// TIA Portal project "LMBMD_ModbusDeviceRtu_0.0.2" (V15.1)

(* hardware
DEVICE "S7-1200 station_1"  S7-1200 Station
   slot 0: "Rack_0"  S7-1200 Rack  Rack  V1.0
   slot 1: "PLC_1"  CPU 1214C DC/DC/DC  6ES7 214-1AG40-0XB0  V4.3
   slot 3: "CB1"  CB 1241 (RS485)  6ES7 241-1CH30-1XB0  V1.0
*)

// ===== PLC "PLC_1"  CPU 1214C DC/DC/DC =====

VAR_GLOBAL   // PLC tag table "Default tag table"
   "System_Byte" AT %MB500 : Byte;
   "FirstScan" AT %M500.0 : Bool;
   "DiagStatusUpdate" AT %M500.1 : Bool;
   "AlwaysTRUE" AT %M500.2 : Bool;
   "AlwaysFALSE" AT %M500.3 : Bool;
   "System_Byte(1)" AT %MB1 : Byte;
   "System_Byte(2)" AT %MB1 : Byte;
   "Clock_Byte" AT %MB501 : Byte;
   "Clock_10Hz" AT %M501.0 : Bool;
   "Clock_5Hz" AT %M501.1 : Bool;
   "Clock_2.5Hz" AT %M501.2 : Bool;
   "Clock_2Hz" AT %M501.3 : Bool;
   "Clock_1.25Hz" AT %M501.4 : Bool;
   "Clock_1Hz" AT %M501.5 : Bool;
   "Clock_0.625Hz" AT %M501.6 : Bool;
   "Clock_0.5Hz" AT %M501.7 : Bool;
END_VAR

// folder: Example

TYPE "DeviceData"
   STRUCT
      param1 : Word;
      param2 : Word;
   END_STRUCT;
END_TYPE

// folder: LMBMD_ModbusDeviceRtu_Master

TYPE "LMBMD_ModbusDeviceRtu_RequestCfg"
// Modbus request configuration
   STRUCT
      mode : USInt := 0;   // Mode / Режим опроса
      dataAddr : UDInt := 40001;   // Starting address in the slave / Начальный адрес регистра
      len : UInt := 1;   // Data length / Длина запроса
      mapAddr : DInt := 0;   // Starting address in the read/write buffer
      enable : Bool := false;   // Заблокировать запрос / Enable request
   END_STRUCT;
END_TYPE

TYPE "LMBMD_ModbusDeviceRtu_Request"
   STRUCT
      cfg : "LMBMD_ModbusDeviceRtu_RequestCfg";
      status : "LMBMD_ModbusDeviceRtu_RequestStatus";
   END_STRUCT;
END_TYPE

TYPE "LMBMD_ModbusDeviceRtu_Data"
   STRUCT
      address : UInt;   // Modbus RTU station address
      buffer : Array[0..100] of Word;
      requests : Array[0..9] of "LMBMD_ModbusDeviceRtu_Request";
   END_STRUCT;
END_TYPE

TYPE "LMBMD_ModbusDeviceRtu_RequestStatus"
// Modbus request status
   STRUCT
      req : Bool;   // Команда на отпарвку запроса
      done : Bool;   // Опрос завершен
      busy : Bool;   // Блок в работе
      error : Bool;   // Ошибка
      status : Word;   // Статус / Error code
      errorCounter : UInt;
   END_STRUCT;
END_TYPE

TYPE "LMBMD_ModbusDeviceRtu_ComPortData"
TITLE = Настройки COM-порта
// Настройки COM-порта
   STRUCT
      port : Port := 271;   // ID порта / ID Port
      baud : UDInt := 9600;   // Скорость / Baudrate
      parity : UInt := 2;   // Паритет (0 - Нет, 1 - Нечет, 2 - Чет ) / Parity (0- None, 1 - Odd, 2 - Even)
      stopBits : UInt;   // Number of stop bits per character Valid values 1 and 2
      timeout : UInt := 500;   // Максимальное время ответа / Response timeout, ms
      status : Word;   // Статус / Response timeout
      done : Bool;   // Инициализация завершена / Execution of instruction completed without error
      error : Bool;   // Ошибка инициализации / Error
      retries : Word := 2;   // Количество повторных запросово / The number of repeated attempts by the master before the error code 0x80C8 is returned for "No response
   END_STRUCT;
END_TYPE

// folder: Example/Data

DATA_BLOCK "DataDb"   // DB1
{ S7_Optimized_Access := 'TRUE' }
VERSION : 0.1
   VAR
      device : "DeviceData";
   END_VAR
BEGIN
END_DATA_BLOCK

DATA_BLOCK "ModbusRtuMaster_DevicesDb"   // DB2
{ S7_Optimized_Access := 'TRUE' }
VERSION : 0.1
   VAR
      device1 : "LMBMD_ModbusDeviceRtu_Data";   // Device 1
      device2 : "LMBMD_ModbusDeviceRtu_Data";   // Device 2
   END_VAR
BEGIN
   device1.address := 1;
   device1.requests[0].cfg.mode := 0;
   device1.requests[0].cfg.dataAddr := 40001;
   device1.requests[0].cfg.len := 2;
   device1.requests[0].cfg.mapAddr := 0;
   device1.requests[0].cfg.enable := true;
   device1.requests[1].cfg.enable := TRUE;
   device1.requests[1].cfg.mapAddr := 1;
   device1.requests[1].cfg.len := 1;
   device2.requests[0].cfg.mapAddr := 0;
   device2.requests[0].cfg.mode := 1;
   device2.requests[0].cfg.dataAddr := 40003;
   device1.requests[1].cfg.dataAddr := 40002;
   device1.requests[1].cfg.mode := 0;
   device2.requests[0].cfg.len := 2;
   device2.address := 2;
   device2.requests[0].cfg.enable := true;
   device1.requests[9].cfg.enable := false;
   device1.requests[9].cfg.mapAddr := 0;
   device1.requests[9].cfg.len := 1;
   device1.requests[9].cfg.dataAddr := 40001;
   device1.requests[9].cfg.mode := 0;
END_DATA_BLOCK

// folder: Example/Inst

DATA_BLOCK "inst_ModbusRtu_Master"   // DB3
{ S7_Optimized_Access := 'TRUE' }
VERSION : 0.1
// stored: InstanceOfName ModbusRtu_Master
"ModbusRtu_Master"
BEGIN
END_DATA_BLOCK

// folder: LMBMD_ModbusDeviceRtu/Data

DATA_BLOCK "LMBMD_ModbusDeviceRtu_CfgDb"   // DB21
{ S7_Optimized_Access := 'TRUE' }
AUTHOR : Veshtemov
VERSION : 0.1
// Конфигурация регистров чтения по Modbus RTU
   VAR
      com : "LMBMD_ModbusDeviceRtu_ComPortData";
   END_VAR
BEGIN
   com.port := 269;
   com.baud := 9600;
   com.retries := 1;
   com.parity := 2;
   com.stopBits := 1;
END_DATA_BLOCK

DATA_BLOCK "LMBMD_ModbusDeviceRtu_DataDb"   // DB24
{ S7_Optimized_Access := 'FALSE' }
VERSION : 0.1
   VAR
      readBuffer : Array[0..255] of Byte;
      writeBuffer : Array[0..255] of Byte;
   END_VAR
BEGIN
END_DATA_BLOCK

// folder: Example

ORGANIZATION_BLOCK "Main"   // OB1, SCL, ProgramCycle
TITLE = "Main Program Sweep (Cycle)"
{ S7_Optimized_Access := 'TRUE' }
VERSION : 0.1
   VAR_INPUT
      Initial_Call : Bool;   // Initial call of this OB
      Remanence : Bool;   // =True, if remanent data are available
   END_VAR
BEGIN
   "inst_ModbusRtu_Master"(com:="LMBMD_ModbusDeviceRtu_CfgDb".com,
                           mbCommLoad:="Modbus_Comm_Load_DB",
                           mbMaster:="Modbus_Master_DB");
END_ORGANIZATION_BLOCK

// folder: Example/RS485/ModbusRtuMaster

FUNCTION_BLOCK "ModbusRtu_Master"   // FB5, SCL
{ S7_Optimized_Access := 'TRUE' }
VERSION : 0.1
// Modbus Rtu Bus
   VAR_IN_OUT
      com : "LMBMD_ModbusDeviceRtu_ComPortData";   // Serial port settings
      mbCommLoad : Modbus_Comm_Load;   // Instance of "Modbus_Comm_Load" function block
      mbMaster : Modbus_Master;   // Instance of "Modbus_Master" function block
   END_VAR
   VAR
      initTrig : R_TRIG;
      inst_LModbusDeviceRtu_Master : "LMBMD_ModbusDeviceRtu_Master";
      i : UInt;
      start : Bool;
   END_VAR
BEGIN
   // Modbus RTU Master

   REGION Serial port initialization
       IF "FirstScan" THEN
           #mbCommLoad.MODE := 4;
       END_IF;

       #mbCommLoad.RETRIES := #com.retries;

       #mbCommLoad(REQ := "FirstScan",
                   "PORT" := #com."port",
                   BAUD := #com.baud,
                   PARITY := #com.parity,
                   MB_DB := #mbMaster.MB_DB,
                   RESP_TO := #com.timeout,
                   DONE => #com.done,
                   ERROR => #com.error,
                   STATUS => #com.status);

       #initTrig(CLK := #com.done);

       IF #initTrig.Q THEN
           #i := 0;
       END_IF;
   END_REGION

   #start := NOT #inst_LModbusDeviceRtu_Master.done;

   CASE #i OF
       0:  // Device 1

           "ModbusRtu_Device1_MapData"(mdata := "ModbusRtuMaster_DevicesDb".device1,
                                       data := "DataDb".device);

           #inst_LModbusDeviceRtu_Master(start := #start,
                                         readBuffer := "LMBMD_ModbusDeviceRtu_DataDb".readBuffer,
                                         writeBuffer := "LMBMD_ModbusDeviceRtu_DataDb".writeBuffer,
                                         data := "ModbusRtuMaster_DevicesDb".device1,
                                         mbMaster := #mbMaster);

           IF #inst_LModbusDeviceRtu_Master.done THEN
               #i := #i + 1;
           END_IF;

       1:  // Device 2
           "ModbusRtu_Device2_MapData"(mdata := "ModbusRtuMaster_DevicesDb".device2,
                                       data := "DataDb".device);

           #inst_LModbusDeviceRtu_Master(start := #start,
                                         readBuffer := "LMBMD_ModbusDeviceRtu_DataDb".readBuffer,
                                         writeBuffer := "LMBMD_ModbusDeviceRtu_DataDb".writeBuffer,
                                         data := "ModbusRtuMaster_DevicesDb".device2,
                                         mbMaster := #mbMaster);

           IF #inst_LModbusDeviceRtu_Master.done THEN
               #i := #i + 1;
           END_IF;
       ELSE
           #i := 0;
   END_CASE;
END_FUNCTION_BLOCK

FUNCTION "ModbusRtu_Device2_MapData" : Void   // FC1, SCL
{ S7_Optimized_Access := 'TRUE' }
VERSION : 0.1
   VAR_IN_OUT
      mdata : "LMBMD_ModbusDeviceRtu_Data";
      data : "DeviceData";
   END_VAR
BEGIN
   // Data
   #mdata.buffer[0] := #data.param1;
   #mdata.buffer[1] := #data.param2;
END_FUNCTION

FUNCTION "ModbusRtu_Device1_MapData" : Void   // FC18, SCL
{ S7_Optimized_Access := 'TRUE' }
VERSION : 0.1
   VAR_IN_OUT
      mdata : "LMBMD_ModbusDeviceRtu_Data";
      data : "DeviceData";
   END_VAR
BEGIN
   // Data
   #data.param1 := #mdata.buffer[0];
   #data.param2 := #mdata.buffer[1];
END_FUNCTION

// folder: LMBMD_ModbusDeviceRtu/Core

FUNCTION_BLOCK "LMBMD_ModbusDeviceRtu_Master"   // FB7, SCL
{ S7_Optimized_Access := 'TRUE' }
VERSION : 0.1
   VAR_INPUT
      start : Bool;   // Пуск / Start block
   END_VAR
   VAR_OUTPUT
      busy : Bool;   // В процессе / In progress
      done : Bool;   // Окончание / Done
   END_VAR
   VAR_IN_OUT
      readBuffer : Variant;   // Буфер обмена / Pointer of read buffer (non optimized data block). For example, DB -> readBuffer: Array[0..125] of Word
      writeBuffer : Variant;   // Pointer of write buffer (non optimized data block). For example, DB -> writeBuffer: Array[0..125] of Word
      data : "LMBMD_ModbusDeviceRtu_Data";
      mbMaster : Modbus_Master;   // Instance of Modbus_Master function block
   END_VAR
   VAR
      buffer : Array[0..127] of Word;
      inst_startTrig : R_TRIG;   // Detect start
      inst_watchdogTimer : TON_TIME;   // Timer for resetting a request when unknown reason is happened
      state : USInt;   // Текущая стадия обмена / Current state
      i : Int;
      j : Int;
   END_VAR
   VAR_TEMP
      tempStart : Bool;   // Start flag
      tempRetval : Int;
      tempQntRequests : Int;   // Quantity of requests
      tempZeroIndex : DInt;
   END_VAR
   VAR CONSTANT
      STATE_STANDBY : USInt := 0;   // Ожидание / State. Standby
      STATE_SETTINGS : USInt := 1;   // Конфигурирование запроса / State. Get settings
      STATE_READ : USInt := 2;   // Запрос на чтение / State. Reading
      STATE_WRITE : USInt := 3;   // Запрос на запись / State. Writing
      STATE_HANDLE : USInt := 4;   // Обработка запроса / State. Handle results
      WATCHDOG_TIME : Time := T#10S;   // Максимальное время ожидания / Watchdog time
      ERROR_ILLEGAL_REQUEST : Word := 16#9000;   // Error. Illegal request (check request settings)
      ERROR_WATCHDOG_TIMER : Word := 16#9001;   // Error. Watchdog timer
   END_VAR
BEGIN
   #tempQntRequests := UDINT_TO_INT("LMBMD_ModbusDeviceRtu_GetArrayLength"(arr := #data.requests));
   #busy := (#state > #STATE_STANDBY); // Set busy flag

   #inst_startTrig(CLK := #start, Q => #tempStart);

   // When start go to Settings
   IF #tempStart THEN

       #done := false;
       #state := #STATE_SETTINGS;

   END_IF;

   CASE #state OF

       // Standby
       #STATE_STANDBY:

           #done := false;
           #i := 0;

       // Get request settings
       #STATE_SETTINGS:

           // With the first call we reset the counter, get the first request,
           // else we increase counter by 1 and get a next request
           IF #tempStart THEN
               #i := 0;

           ELSE
               #i := #i + 1;

               // When all requests is completed go to standby, set "done" flag 
               IF #i >= #tempQntRequests THEN
                   #done := true;
                   #state := #STATE_STANDBY;
                   RETURN;
               END_IF;
           END_IF;

           // Check request settings: we have to skip disabled or invalid requests,
           // if a request is invalid - set ERROR_ILLEGAL_REQUEST status
           FOR #j := #i TO #tempQntRequests - 1 DO

               IF NOT #data.requests[#j].cfg.enable THEN

                   #data.requests[#j].status.req := false;
                   #data.requests[#j].status.done := false;
                   #data.requests[#j].status.error := false;
                   #data.requests[#j].status.status := 0;
                   #data.requests[#j].status.errorCounter := 0;

               ELSIF NOT "LMBMD_ModbusDeviceRtu_ValidateRequest"(#data.requests[#j].cfg) THEN

                   // Set error status
                   #data.requests[#j].status.req := false;
                   #data.requests[#j].status.done := false;
                   #data.requests[#j].status.error := true;
                   #data.requests[#j].status.status := #ERROR_ILLEGAL_REQUEST;
                   #data.requests[#j].status.errorCounter := LIMIT(IN := #data.requests[#j].status.errorCounter + 1,
                                                                   MN := 0,
                                                                   MX := 65534);
               ELSE
                   #i := #j;
                   EXIT;
               END_IF;

               // When all requests is completed go to standby, set "done" flag
               IF #j = #tempQntRequests - 1 THEN
                   #done := true;
                   #state := #STATE_STANDBY;
                   RETURN;
               END_IF;

           END_FOR;

           // For writing before request we have to copy data to external write buffer
           IF #data.requests[#i].cfg.mode > 0 THEN

               // Extract data from Modbus Device to write buffer
               MOVE_BLK(IN := #data.#buffer[#data.requests[#i].cfg.mapAddr],
                        COUNT := #data.requests[#i].cfg.len,
                        OUT => #buffer[0]);

               #tempZeroIndex := 0;
               #tempRetval := Serialize(SRC_VARIABLE := #buffer,
                                        DEST_ARRAY => #writeBuffer,
                                        POS := #tempZeroIndex);

               #state := #STATE_WRITE;
           ELSE
               #state := #STATE_READ;
           END_IF;

           RETURN;

       // Read
       #STATE_READ, #STATE_WRITE:

           #data.requests[#i].status.req := true;

       // Handle results
       #STATE_HANDLE:

           #data.requests[#i].status.req := false;

           IF #data.requests[#i].status.done THEN
               #data.requests[#i].status.errorCounter := 0;

               // Copy from modbus buffer to device buffer
               IF #data.requests[#i].cfg.mode = 0 THEN

                   #tempZeroIndex := 0;
                   #tempRetval := Deserialize(SRC_ARRAY := #readBuffer,
                                              DEST_VARIABLE => #buffer,
                                              POS := #tempZeroIndex);
                   MOVE_BLK(IN := #buffer[0],
                            COUNT := #data.requests[#i].cfg.len,
                            OUT => #data.buffer[#data.requests[#i].cfg.mapAddr]);
               END_IF;

           ELSIF #data.requests[#i].status.error THEN
               #data.requests[#i].status.errorCounter := LIMIT(IN := #data.requests[#i].status.errorCounter + 1,
                                                               MN := 0,
                                                               MX := 65534);
           END_IF;

           #state := #STATE_SETTINGS;

       ELSE
           #state := #STATE_STANDBY;
   END_CASE;

   // There are different buffers for reading and writing
   IF (#state = #STATE_READ) THEN
       // Request
       #mbMaster(REQ := #data.requests[#i].status.req,
                 MB_ADDR := #data.address,
                 MODE := #data.requests[#i].cfg.mode,
                 DATA_ADDR := #data.requests[#i].cfg.dataAddr,
                 DATA_LEN := #data.requests[#i].cfg.len,
                 DONE => #data.requests[#i].status.done,
                 BUSY => #data.requests[#i].status.busy,
                 ERROR => #data.requests[#i].status.error,
                 STATUS => #data.requests[#i].status.status,
                 DATA_PTR := #readBuffer);

   ELSIF (#state = #STATE_WRITE) THEN
       // Запрос
       #mbMaster(REQ := #data.requests[#i].status.req,
                 MB_ADDR := #data.address,
                 MODE := #data.requests[#i].cfg.mode,
                 DATA_ADDR := #data.requests[#i].cfg.dataAddr,
                 DATA_LEN := #data.requests[#i].cfg.len,
                 DONE => #data.requests[#i].status.done,
                 BUSY => #data.requests[#i].status.busy,
                 ERROR => #data.requests[#i].status.error,
                 STATUS => #data.requests[#i].status.status,
                 DATA_PTR := #writeBuffer);
   END_IF;


   // Waiting response status
   IF ((#state = #STATE_READ
       OR #state = #STATE_WRITE)
       AND (#data.requests[#i].status.done
       OR #data.requests[#i].status.error))
   THEN
       #state := #STATE_HANDLE;
   END_IF;

   // Watchdog timer is needed when state stuck in Read or Write state for unknown reason,
   // in that case we set request as invalid 
   #inst_watchdogTimer(IN := (#state = #STATE_READ
                  OR #state = #STATE_WRITE),
                  PT := #WATCHDOG_TIME);

   IF #inst_watchdogTimer.Q THEN

       #data.requests[#i].status.done := false;
       #data.requests[#i].status.error := true;
       #data.requests[#i].status.status := #ERROR_WATCHDOG_TIMER;
       #data.requests[#i].status.errorCounter := LIMIT(IN := #data.requests[#i].status.errorCounter + 1,
                                                       MN := 0,
                                                       MX := 65534);

       #state := #STATE_HANDLE;

   END_IF;
END_FUNCTION_BLOCK

FUNCTION "LMBMD_ModbusDeviceRtu_ValidateRequest" : Bool   // FC2, SCL
{ S7_Optimized_Access := 'TRUE' }
VERSION : 0.1
   VAR_IN_OUT
      data : "LMBMD_ModbusDeviceRtu_RequestCfg";
   END_VAR
BEGIN
   #LMBMD_ModbusDeviceRtu_ValidateRequest :=
   #data.len > 0
   AND (#data.mode >= 0 AND #data.mode <= 2);
END_FUNCTION

FUNCTION "LMBMD_ModbusDeviceRtu_GetArrayLength" : UDInt   // FC9, SCL
{ S7_Optimized_Access := 'TRUE' }
VERSION : 0.1
   VAR_INPUT
      arr : Variant;
   END_VAR
BEGIN
   IF IS_ARRAY(#arr) THEN
       #LMBMD_ModbusDeviceRtu_GetArrayLength := CountOfElements(IN := #arr);
   ELSE
       #LMBMD_ModbusDeviceRtu_GetArrayLength := 0;
   END_IF;
END_FUNCTION

// ===== library: MasterCopy "LMB_ModbusDeviceRtu_Buffer" =====

// folder: LMB_ModbusDeviceRtu_Master

TYPE "LMB_ModbusDeviceRtu_Buffer"
// Raw data of Modbus device
   STRUCT
      readBuffer : Array[0..100] of Word;   // Read buffer
      writeBuffer : Array[0..100] of Word;   // Write buffer
   END_STRUCT;
END_TYPE

// ===== library: MasterCopy "LMB_ModbusDeviceRtu_ComPortData" =====

// folder: LMB_ModbusDeviceRtu_Master

TYPE "LMB_ModbusDeviceRtu_ComPortData"
TITLE = Настройки COM-порта
// Настройки COM-порта
   STRUCT
      port : Port := 271;   // ID порта / ID Port
      baud : UDInt := 9600;   // Скорость / Baudrate
      parity : UInt := 2;   // Паритет (0 - Нет, 1 - Нечет, 2 - Чет ) / Parity (0- None, 1 - Odd, 2 - Even)
      stopBits : UInt;   // Number of stop bits per character Valid values 1 and 2
      timeout : UInt := 500;   // Максимальное время ответа / Response timeout, ms
      status : Word;   // Статус / Response timeout
      done : Bool;   // Инициализация завершена / Execution of instruction completed without error
      error : Bool;   // Ошибка инициализации / Error
      retries : Word := 2;   // Количество повторных запросово / The number of repeated attempts by the master before the error code 0x80C8 is returned for "No response
   END_STRUCT;
END_TYPE

// ===== library: MasterCopy "LMB_ModbusDeviceRtu_Data" =====

// folder: LMB_ModbusDeviceRtu_Master

TYPE "LMB_ModbusDeviceRtu_Data"
   STRUCT
      addresss : UInt;   // Modbus RTU station address
      buffer : "LMB_ModbusDeviceRtu_Buffer";
      requests : Array[0..9] of "LMB_ModbusDeviceRtu_Request";
   END_STRUCT;
END_TYPE

// ===== library: MasterCopy "LMB_ModbusDeviceRtu_Request" =====

// folder: LMB_ModbusDeviceRtu_Master

TYPE "LMB_ModbusDeviceRtu_Request"
   STRUCT
      cfg : "LMB_ModbusDeviceRtu_RequestCfg";
      status : "LMB_ModbusDeviceRtu_RequestStatus";
   END_STRUCT;
END_TYPE

// ===== library: MasterCopy "LMB_ModbusDeviceRtu_RequestCfg" =====

// folder: LMB_ModbusDeviceRtu_Master

TYPE "LMB_ModbusDeviceRtu_RequestCfg"
// Modbus request configuration
   STRUCT
      mode : USInt := 0;   // Mode / Режим опроса
      dataAddr : UDInt := 40001;   // Starting address in the slave / Начальный адрес регистра
      len : UInt := 1;   // Data length / Длина запроса
      mapAddr : DInt := 0;   // Starting address in the read/write buffer
      enable : Bool := false;   // Заблокировать запрос / Enable request
   END_STRUCT;
END_TYPE

// ===== library: MasterCopy "LMB_ModbusDeviceRtu_RequestStatus" =====

// folder: LMB_ModbusDeviceRtu_Master

TYPE "LMB_ModbusDeviceRtu_RequestStatus"
// Modbus request status
   STRUCT
      req : Bool;   // Команда на отпарвку запроса
      done : Bool;   // Опрос завершен
      busy : Bool;   // Блок в работе
      error : Bool;   // Ошибка
      status : Word;   // Статус / Error code
      errorCounter : UInt;
   END_STRUCT;
END_TYPE

// ===== library: MasterCopy "LMB_ModbusDeviceRtu_GetArrayLength" =====

// folder: LMB_ModbusDeviceRtu_Master/Core

FUNCTION "LMB_ModbusDeviceRtu_GetArrayLength" : UDInt   // FC9, SCL
{ S7_Optimized_Access := 'TRUE' }
VERSION : 0.1
   VAR_INPUT
      arr : Variant;
   END_VAR
BEGIN
   IF IS_ARRAY(#arr) THEN
       #LMB_ModbusDeviceRtu_GetArrayLength := CountOfElements(IN := #arr);
   ELSE
       #LMB_ModbusDeviceRtu_GetArrayLength := 0;
   END_IF;
END_FUNCTION

// ===== library: MasterCopy "LMB_ModbusDeviceRtu_ValidateRequest" =====

// folder: LMB_ModbusDeviceRtu_Master/Core

FUNCTION "LMB_ModbusDeviceRtu_ValidateRequest" : Bool   // FC2, SCL
{ S7_Optimized_Access := 'TRUE' }
VERSION : 0.1
   VAR_IN_OUT
      data : "LMB_ModbusDeviceRtu_RequestCfg";
   END_VAR
BEGIN
   #LMB_ModbusDeviceRtu_ValidateRequest :=
   #data.len > 0
   AND (#data.mode >= 0 AND #data.mode <= 2);
END_FUNCTION

// ===== library: MasterCopy "LMB_ModbusDeviceRtu_Master" =====

// folder: LMB_ModbusDeviceRtu_Master/Core

FUNCTION_BLOCK "LMB_ModbusDeviceRtu_Master"   // FB7, SCL
{ S7_Optimized_Access := 'TRUE' }
VERSION : 0.1
   VAR_INPUT
      start : Bool;   // Пуск / Start block
   END_VAR
   VAR_OUTPUT
      busy : Bool;   // В процессе / In progress
      done : Bool;   // Окончание / Done
   END_VAR
   VAR_IN_OUT
      readBuffer : Variant;   // Буфер обмена / Pointer of read buffer (non optimized data block). For example, DB -> readBuffer: Array[0..125] of Word
      writeBuffer : Variant;   // Pointer of write buffer (non optimized data block). For example, DB -> writeBuffer: Array[0..125] of Word
      data : "LMB_ModbusDeviceRtu_Data";
      mbMaster : Modbus_Master;   // Instance of Modbus_Master function block
   END_VAR
   VAR
      inst_startTrig : R_TRIG;   // Detect start
      inst_watchdogTimer : TON_TIME;   // Timer for resetting a request when unknown reason is happened
      state : USInt;   // Текущая стадия обмена / Current state
      i : Int;
      j : Int;
   END_VAR
   VAR_TEMP
      tempStart : Bool;   // Start flag
      tempRetval : Int;
      tempQntRequests : Int;   // Quantity of requests
   END_VAR
   VAR CONSTANT
      STATE_STANDBY : USInt := 0;   // Ожидание / State. Standby
      STATE_SETTINGS : USInt := 1;   // Конфигурирование запроса / State. Get settings
      STATE_READ : USInt := 2;   // Запрос на чтение / State. Reading
      STATE_WRITE : USInt := 3;   // Запрос на запись / State. Writing
      STATE_HANDLE : USInt := 4;   // Обработка запроса / State. Handle results
      WATCHDOG_TIME : Time := T#10S;   // Максимальное время ожидания / Watchdog time
      ERROR_ILLEGAL_REQUEST : Word := 16#8500;   // Error. Illegal request (check request settings)
      ERROR_WATCHDOG_TIMER : Word := 16#8501;   // Error. Watchdog timer
   END_VAR
BEGIN
   #tempQntRequests := UDINT_TO_INT("LMB_ModbusDeviceRtu_GetArrayLength"(arr := #data.requests));
   #busy := (#state > #STATE_STANDBY); // Set busy flag

   #inst_startTrig(CLK := #start, Q => #tempStart);

   // When start go to Settings
   IF #tempStart THEN

       #done := false;
       #state := #STATE_SETTINGS;

   END_IF;

   CASE #state OF

       // Standby
       #STATE_STANDBY:

           #done := false;
           #i := 0;

       // Get request settings
       #STATE_SETTINGS:

           // With the first call we reset the counter, get the first request,
           // else we increase counter by 1 and get a next request
           IF #tempStart THEN
               #i := 0;

           ELSE
               #i := #i + 1;

               // When all requests is completed go to standby, set "done" flag 
               IF #i >= #tempQntRequests THEN
                   #done := true;
                   #state := #STATE_STANDBY;
                   RETURN;
               END_IF;
           END_IF;

           // Check request settings: we have to skip disabled or invalid requests,
           // if a request is invalid - set ERROR_ILLEGAL_REQUEST status
           FOR #j := #i TO #tempQntRequests - 1 DO

               IF NOT #data.requests[#j].cfg.enable THEN

                   #data.requests[#j].status.req := false;
                   #data.requests[#j].status.done := false;
                   #data.requests[#j].status.error := false;
                   #data.requests[#j].status.status := 0;
                   #data.requests[#j].status.errorCounter := 0;

               ELSIF NOT "LMB_ModbusDeviceRtu_ValidateRequest"(#data.requests[#j].cfg) THEN

                   // Set error status
                   #data.requests[#j].status.req := false;
                   #data.requests[#j].status.done := false;
                   #data.requests[#j].status.error := true;
                   #data.requests[#j].status.status := #ERROR_ILLEGAL_REQUEST;
                   #data.requests[#j].status.errorCounter := LIMIT(IN := #data.requests[#j].status.errorCounter + 1,
                                                                   MN := 0,
                                                                   MX := 65534);
               ELSE
                   #i := #j;
                   EXIT;
               END_IF;

               // When all requests is completed go to standby, set "done" flag
               IF #j = #tempQntRequests - 1 THEN
                   #done := true;
                   #state := #STATE_STANDBY;
                   RETURN;
               END_IF;

           END_FOR;

           // For writing before request we have to copy data to external write buffer
           IF #data.requests[#i].cfg.mode > 0 THEN

               // Extract data from Modbus Device write buffer
               #tempRetval := Serialize(SRC_VARIABLE := #data.buffer.writeBuffer,
                                        DEST_ARRAY => #writeBuffer,
                                        POS := #data.requests[#i].cfg.mapAddr);
               #state := #STATE_WRITE;
           ELSE
               #state := #STATE_READ;
           END_IF;

           RETURN;

       // Read
       #STATE_READ, #STATE_WRITE:

           #data.requests[#i].status.req := true;

       // Handle results
       #STATE_HANDLE:

           #data.requests[#i].status.req := false;

           IF #data.requests[#i].status.done THEN
               #data.requests[#i].status.errorCounter := 0;
           ELSIF #data.requests[#i].status.error THEN
               #data.requests[#i].status.errorCounter := LIMIT(IN := #data.requests[#i].status.errorCounter + 1,
                                                               MN := 0,
                                                               MX := 65534);
           END_IF;

           #state := #STATE_SETTINGS;

       ELSE
           #state := #STATE_STANDBY;
   END_CASE;

   // There are different buffers for reading and writing
   IF (#state = #STATE_READ) THEN
       // Request
       #mbMaster(REQ := #data.requests[#i].status.req,
                 MB_ADDR := #data.address,
                 MODE := #data.requests[#i].cfg.mode,
                 DATA_ADDR := #data.requests[#i].cfg.dataAddr,
                 DATA_LEN := #data.requests[#i].cfg.len,
                 DONE => #data.requests[#i].status.done,
                 BUSY => #data.requests[#i].status.busy,
                 ERROR => #data.requests[#i].status.error,
                 STATUS => #data.requests[#i].status.status,
                 DATA_PTR := #readBuffer);

   ELSIF (#state = #STATE_WRITE) THEN
       // Запрос
       #mbMaster(REQ := #data.requests[#i].status.req,
                 MB_ADDR := #data.address,
                 MODE := #data.requests[#i].cfg.mode,
                 DATA_ADDR := #data.requests[#i].cfg.dataAddr,
                 DATA_LEN := #data.requests[#i].cfg.len,
                 DONE => #data.requests[#i].status.done,
                 BUSY => #data.requests[#i].status.busy,
                 ERROR => #data.requests[#i].status.error,
                 STATUS => #data.requests[#i].status.status,
                 DATA_PTR := #writeBuffer);
   END_IF;


   // Waiting response status
   IF ((#state = #STATE_READ
       OR #state = #STATE_WRITE)
       AND (#data.requests[#i].status.done
       OR #data.requests[#i].status.error))
   THEN
       #state := #STATE_HANDLE;
   END_IF;

   // Watchdog timer is needed when state stuck in Read or Write state for unknown reason,
   // in that case we set request as invalid 
   #inst_watchdogTimer(IN := (#state = #STATE_READ
                  OR #state = #STATE_WRITE),
                  PT := #WATCHDOG_TIME);

   IF #inst_watchdogTimer.Q THEN

       #data.requests[#i].status.done := false;
       #data.requests[#i].status.error := true;
       #data.requests[#i].status.status := #ERROR_WATCHDOG_TIMER;
       #data.requests[#i].status.errorCounter := LIMIT(IN := #data.requests[#i].status.errorCounter + 1,
                                                       MN := 0,
                                                       MX := 65534);

       #state := #STATE_HANDLE;

   END_IF;
END_FUNCTION_BLOCK

// ===== library: MasterCopy "LMB_ModbusDeviceRtu_CfgDb" =====

// folder: LMB_ModbusDeviceRtu_Master/Data

DATA_BLOCK "LMB_ModbusDeviceRtu_CfgDb"   // DB21
{ S7_Optimized_Access := 'TRUE' }
AUTHOR : Veshtemov
VERSION : 0.1
// Конфигурация регистров чтения по Modbus RTU
   VAR
      com : "LMB_ModbusDeviceRtu_ComPortData";
   END_VAR
BEGIN
   com.port := 269;
   com.baud := 9600;
   com.retries := 1;
   com.parity := 2;
   com.stopBits := 1;
END_DATA_BLOCK

// ===== library: MasterCopy "LMB_ModbusDeviceRtu_DataDb" =====

// folder: LMB_ModbusDeviceRtu_Master/Data

DATA_BLOCK "LMB_ModbusDeviceRtu_DataDb"   // DB24
{ S7_Optimized_Access := 'FALSE' }
VERSION : 0.1
   VAR
      buffer : Array[0..125] of Word;
      writeBuffer : Array[0..125] of Word;
   END_VAR
BEGIN
END_DATA_BLOCK